// TIA Portal V16 export
// export: Created 2025-05-30T16:30:17.577149Z, ExportSetting WithDefaults, DisplayName Totally Integrated Automation Portal, DisplayVersion V16, DisplayName TIA Portal Version Control Interface, DisplayVersion V16, DisplayName TIA Portal Openness, DisplayVersion V16, DisplayName STEP 7 Professional, DisplayVersion V16, DisplayName STEP 7 Safety, DisplayVersion V16, DisplayName WinCC Advanced, DisplayVersion V16
FUNCTION "SystemRUN_Block" : Void   // FC13, LAD
VERSION : 0.1
// stored: AutoNumber true, IsIECCheckEnabled false, UDAEnableTagReadback false
   VAR_INPUT
      "Safety Relais Contact" : Bool;
      "Stop Machine NC Contact" : Bool;
      "Fill Magzine Contact" : Bool;
      "Start Machine NO Contact" : Bool;
   END_VAR
   VAR_OUTPUT
      "Run Output Lamp" : Bool;
   END_VAR
BEGIN

REGION Network 1: Systeem RUN
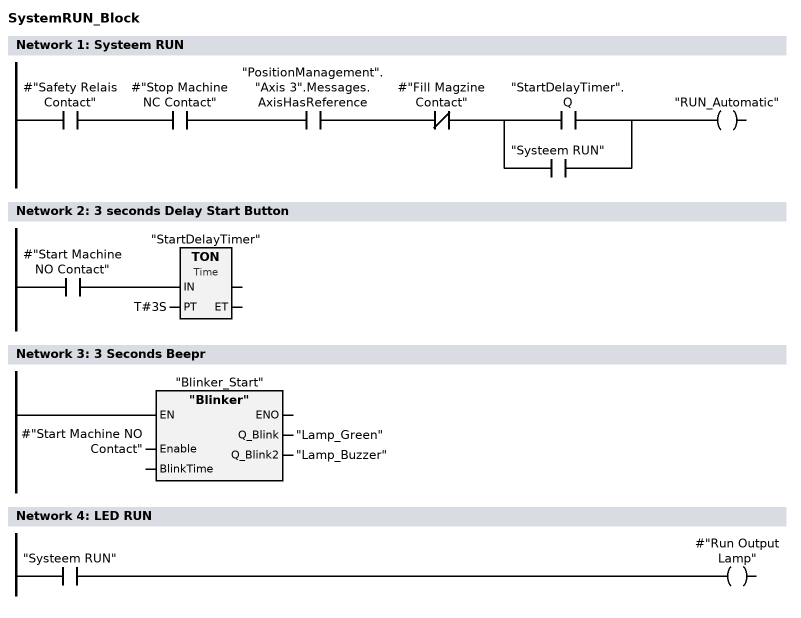
   RUNG wire#powerrail
      Contact( #"Safety Relais Contact" )
      Contact( #"Stop Machine NC Contact" )
      Contact( "PositionManagement"."Axis 3".Messages.AxisHasReference )
      I_Contact( #"Fill Magzine Contact" )
      wire#w1
      Contact( "StartDelayTimer".Q )
      wire#w2
      Coil( "RUN_Automatic" )
   END_RUNG
   RUNG wire#w1
      Contact( "Systeem RUN" )
   END_RUNG wire#w2
   // the same network as SCL:
   "RUN_Automatic" := #"Safety Relais Contact" AND #"Stop Machine NC Contact" AND "PositionManagement"."Axis 3".Messages.AxisHasReference AND NOT #"Fill Magzine Contact" AND ("StartDelayTimer".Q OR "Systeem RUN");
END_REGION

REGION Network 2: 3 seconds Delay Start Button
   RUNG wire#powerrail
      Contact( #"Start Machine NO Contact" )
      { S7_Templates := "time_type := Time" } "StartDelayTimer".TON(pt := T#3S, et =>)
   END_RUNG
   // the same network as SCL:
   "StartDelayTimer".TON(IN := #"Start Machine NO Contact", PT := T#3S);
END_REGION

REGION Network 3: 3 Seconds Beepr
   RUNG wire#powerrail
      "Blinker_Start"(Enable := #"Start Machine NO Contact", BlinkTime :=, Q_Blink => "Lamp_Green", Q_Blink2 => "Lamp_Buzzer")
   END_RUNG
   // the same network as SCL:
   "Blinker_Start"(Enable := #"Start Machine NO Contact", Q_Blink => "Lamp_Green", Q_Blink2 => "Lamp_Buzzer");   // "Blinker"
END_REGION

REGION Network 4: LED RUN
   RUNG wire#powerrail
      Contact( "Systeem RUN" )
      Coil( #"Run Output Lamp" )
   END_RUNG
   // the same network as SCL:
   #"Run Output Lamp" := "Systeem RUN";
END_REGION
END_FUNCTION
